(* IEC 61131-3 sources: eCockpitGit/test_project/src/%F%00 Library/%F%JSON/%POU%FB_JSONReader/%F%Structure/%PRO%selectedType, 1 file *)

(* ---- %GETSET%Get.st ---- *)
VAR
END_VAR

(*%!%__DELIMITER__%!%*)
IF treeLevel > 0 THEN
	selectedType		:=		treeSelectedTypes[treeLevel];
ELSE
	selectedType		:=		buttomType;
END_IF
